// TIA Portal V19 export
DATA_BLOCK "CoilHandlingMatCounter"   // DB205
{ DB_Accessible_From_OPC_UA := 'FALSE' }
// stored: DBAccessibleFromOPCUA false, InstanceOfName MatCounter, InstanceOfType FB
"MatCounter"
   // VAR_INPUT
   //    CIn : "MatCountCIn";
   //    StandstillVelocityThreshold : LReal;
   //    Config : Struct
   //       Default_FAK : LReal;
   //    END_STRUCT;
   // END_VAR
   // VAR_OUTPUT
   //    COut : Struct
   //       AlarmsPresence : Bool;
   //       WarningsPresence : Bool;
   //       StopFeeding : Bool;
   //       CounterValid : Bool;
   //       Standstill : Bool;
   //       PresetDone : Bool;
   //       ActualVelocity : LReal;
   //    END_STRUCT;
   //    Alr : Struct
   //       CounterNotInOperation : Bool;
   //    END_STRUCT;
   //    Wng : Struct
   //       EncoderNotValid : Bool;
   //       EncoderPosNotValid : Bool;
   //       PresetRunning : Bool;
   //    END_STRUCT;
   // END_VAR
   // VAR_IN_OUT
   //    PersistentValues : "MatCountPersistent";
   // END_VAR
   // VAR
   //    Status : Int;
   //    Sts : Struct
   //       PLCStartUpDone : Bool;
   //       Initialization : Bool;
   //       InOperation : Bool;
   //       PresetDone : Bool;
   //       FAKCalcDoneAndApply : Bool;
   //       RestorePreviousFAKDone : Bool;
   //       FAKManChangeApply : Bool;
   //       SetDefaultFAKDone : Bool;
   //       FAKManChange : Bool;
   //       HMIOperationDone : Bool;
   //       NewPositionToForce : LReal;
   //       NewFAK : LReal;
   //       VelocityLessThanThreshold : Bool;
   //    END_STRUCT;
   //    tonInOperation : TON_TIME;
   //    tonOpDone : TON_TIME;
   //    HMI : Struct
   //       PbFAKCalculation : Bool;
   //       PbFAKDefault : Bool;
   //       PbFAKPrevious : Bool;
   //       FAKSetDefaultDone : Bool;
   //       FAKCalcDone : Bool;
   //       FAKSetPrevDone : Bool;
   //       LenghtDesired : LReal;
   //       LenghtMeasured : LReal;
   //       FAKPrevious : LReal;
   //       FAKDefault : LReal;
   //    END_STRUCT;
   //    Aux : Struct
   //       PbFAKCalculation : Bool;
   //       PbFAKDefault : Bool;
   //       PbFAKPrevious : Bool;
   //    END_STRUCT;
   //    Check_Velocity { S7_SetPoint := 'True'} : "Check_Axis_Velocity";
   // END_VAR
BEGIN
END_DATA_BLOCK
